TYPE ST_ContentOUT2 :
STRUCT
	DefaultIdentity   :ST_DefaultIdentityOUT2;
	ExpectedItemCount	:STRING;
	ItemReadRate		:STRING;
	ItemList			:ST_ItemListOUT2;
END_STRUCT
END_TYPE

(* stored: Version 1.1.0.1, ProductVersion 3.1.4024.13
   DUT ST_ContentOUT2: Id {5f20f260-060a-4b28-9a67-86048a84f4a4} *)
